{attribute 'linkalways'}
{attribute 'no_explicit_call' := 'do not call this POU directly'}
FUNCTION_BLOCK ABSTRACT Event IMPLEMENTS I_Event
VAR
	subscribers : SubscriberCollection;
END_VAR

METHOD PUBLIC AddSubscriber
VAR_INPUT
	Subscriber : I_Subscriber;
END_VAR
subscribers.Insert(Subscriber);
END_METHOD

METHOD PROTECTED NotifySubscribers
VAR
	count : UDINT;
	i : UDINT;
END_VAR
count := subscribers.Count;
FOR i := 0 TO count - 1 DO
	subscribers.GetByIndex(i).Update(THIS^);
END_FOR
END_METHOD

METHOD PUBLIC RemoveSubscriber
VAR_INPUT
	Subscriber : I_Subscriber;
END_VAR
subscribers.Remove(Subscriber);
END_METHOD

END_FUNCTION_BLOCK

(* stored: Version 1.1.0.1, ProductVersion 3.1.4024.11
   POU Event: Id {4d0749e9-dd51-4254-8072-025c2ed16feb}, SpecialFunc None
   Folder Protected: Id {f81292ce-63c9-42a8-9fd5-6142ce702b35}
   Method AddSubscriber: Id {dc1fa9a8-111d-4d13-a70c-ecbec31b1df1}
   Method NotifySubscribers: Id {00f6e4c5-1f92-4c04-90a4-78cbf5e7a24d}
   Method RemoveSubscriber: Id {3a25e12d-9cea-4c90-88a9-76f17d36e0cf} *)
